PROGRAM MAIN
VAR
END_VAR

END_PROGRAM

(* stored: Version 1.1.0.1, ProductVersion 3.1.4022.18
   POU MAIN: Id {e5334f36-3c5f-4553-b6cf-4e9240a43836}, SpecialFunc None *)
